// TIA Portal V16 export
// export: Created 2023-08-28T09:37:57.0218965Z, ExportSetting WithDefaults, DisplayName Totally Integrated Automation Portal, DisplayVersion V16 Update 6, DisplayName TIA Portal Version Control Interface, DisplayVersion V16 Update 2, DisplayName TIA Portal Openness, DisplayVersion V16 Update 6, DisplayName STEP 7 Professional, DisplayVersion V16 Update 6, DisplayName STEP 7 Safety, DisplayVersion V16, DisplayName WinCC Advanced, DisplayVersion V16 Update 6
TYPE "typeDataMPP04_int_1"
// stored: IsFailsafeCompliant false
   STRUCT
      data : Array[0..0] of Int;
   END_STRUCT;
END_TYPE
